PROGRAM C25_MC2AxisDriversCtrl
VAR
	fbMC2AxisCtrl		:  FB_MC2_AX5000AxisCtrl;

	stAxisConfig		: ST_AXIS_Config;	(*Has to be defined in Machine Config structure to retain data*)

	bStationHomed		: BOOL;
	bSeqHomingRequest	: BOOL;
	bSeqInProgress		: BOOL;

(*dummy sturcture to be replaced by global MC struct once implemnted*)
{library private}
	nAxis00TorqueLimitation								: UINT	:=	32767;
	nAxis00ActualTorque								 : INT;
	refAxis00											: AXIS_REF;
END_VAR

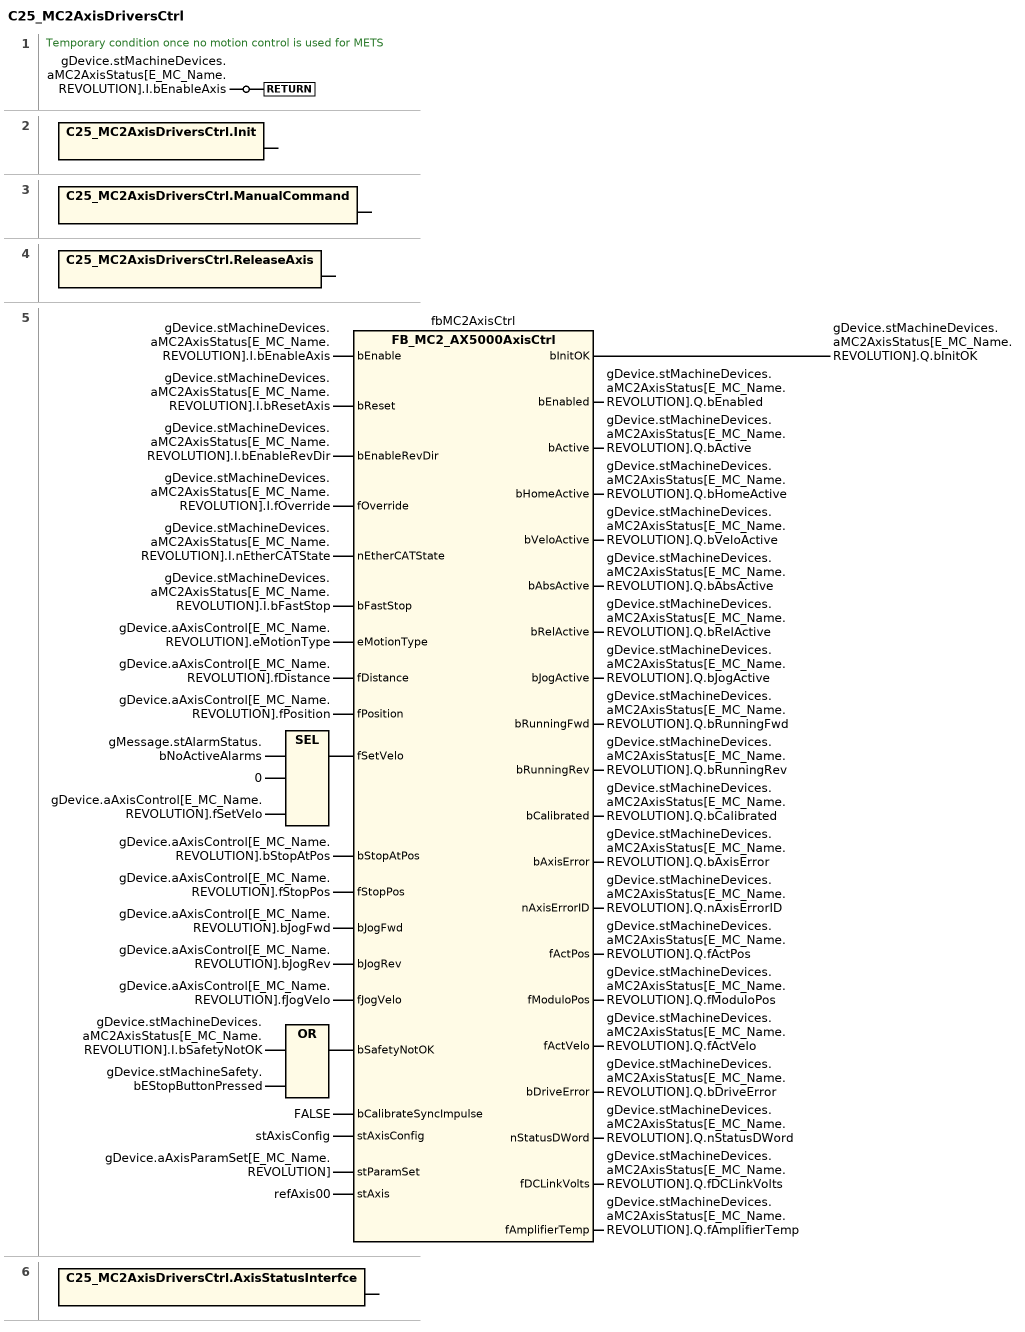
// NETWORK 1
// Temporary condition once no motion control is used for METS
IF NOT gDevice.stMachineDevices.aMC2AxisStatus[E_MC_Name.REVOLUTION].I.bEnableAxis THEN RETURN; END_IF

// NETWORK 2
C25_MC2AxisDriversCtrl.Init();

// NETWORK 3
C25_MC2AxisDriversCtrl.ManualCommand();

// NETWORK 4
C25_MC2AxisDriversCtrl.ReleaseAxis();

// NETWORK 5
fbMC2AxisCtrl(
    bEnable := gDevice.stMachineDevices.aMC2AxisStatus[E_MC_Name.REVOLUTION].I.bEnableAxis,
    bReset := gDevice.stMachineDevices.aMC2AxisStatus[E_MC_Name.REVOLUTION].I.bResetAxis,
    bEnableRevDir := gDevice.stMachineDevices.aMC2AxisStatus[E_MC_Name.REVOLUTION].I.bEnableRevDir,
    fOverride := gDevice.stMachineDevices.aMC2AxisStatus[E_MC_Name.REVOLUTION].I.fOverride,
    nEtherCATState := gDevice.stMachineDevices.aMC2AxisStatus[E_MC_Name.REVOLUTION].I.nEtherCATState,
    bFastStop := gDevice.stMachineDevices.aMC2AxisStatus[E_MC_Name.REVOLUTION].I.bFastStop,
    eMotionType := gDevice.aAxisControl[E_MC_Name.REVOLUTION].eMotionType,
    fDistance := gDevice.aAxisControl[E_MC_Name.REVOLUTION].fDistance,
    fPosition := gDevice.aAxisControl[E_MC_Name.REVOLUTION].fPosition,
    fSetVelo := SEL(gMessage.stAlarmStatus.bNoActiveAlarms, 0, gDevice.aAxisControl[E_MC_Name.REVOLUTION].fSetVelo),
    bStopAtPos := gDevice.aAxisControl[E_MC_Name.REVOLUTION].bStopAtPos,
    fStopPos := gDevice.aAxisControl[E_MC_Name.REVOLUTION].fStopPos,
    bJogFwd := gDevice.aAxisControl[E_MC_Name.REVOLUTION].bJogFwd,
    bJogRev := gDevice.aAxisControl[E_MC_Name.REVOLUTION].bJogRev,
    fJogVelo := gDevice.aAxisControl[E_MC_Name.REVOLUTION].fJogVelo,
    bSafetyNotOK := gDevice.stMachineDevices.aMC2AxisStatus[E_MC_Name.REVOLUTION].I.bSafetyNotOK OR gDevice.stMachineSafety.bEStopButtonPressed,
    bCalibrateSyncImpulse := FALSE,
    stAxisConfig := stAxisConfig,
    stParamSet := gDevice.aAxisParamSet[E_MC_Name.REVOLUTION],
    stAxis := refAxis00,
    bEnabled => gDevice.stMachineDevices.aMC2AxisStatus[E_MC_Name.REVOLUTION].Q.bEnabled,
    bActive => gDevice.stMachineDevices.aMC2AxisStatus[E_MC_Name.REVOLUTION].Q.bActive,
    bHomeActive => gDevice.stMachineDevices.aMC2AxisStatus[E_MC_Name.REVOLUTION].Q.bHomeActive,
    bVeloActive => gDevice.stMachineDevices.aMC2AxisStatus[E_MC_Name.REVOLUTION].Q.bVeloActive,
    bAbsActive => gDevice.stMachineDevices.aMC2AxisStatus[E_MC_Name.REVOLUTION].Q.bAbsActive,
    bRelActive => gDevice.stMachineDevices.aMC2AxisStatus[E_MC_Name.REVOLUTION].Q.bRelActive,
    bJogActive => gDevice.stMachineDevices.aMC2AxisStatus[E_MC_Name.REVOLUTION].Q.bJogActive,
    bRunningFwd => gDevice.stMachineDevices.aMC2AxisStatus[E_MC_Name.REVOLUTION].Q.bRunningFwd,
    bRunningRev => gDevice.stMachineDevices.aMC2AxisStatus[E_MC_Name.REVOLUTION].Q.bRunningRev,
    bCalibrated => gDevice.stMachineDevices.aMC2AxisStatus[E_MC_Name.REVOLUTION].Q.bCalibrated,
    bAxisError => gDevice.stMachineDevices.aMC2AxisStatus[E_MC_Name.REVOLUTION].Q.bAxisError,
    nAxisErrorID => gDevice.stMachineDevices.aMC2AxisStatus[E_MC_Name.REVOLUTION].Q.nAxisErrorID,
    fActPos => gDevice.stMachineDevices.aMC2AxisStatus[E_MC_Name.REVOLUTION].Q.fActPos,
    fModuloPos => gDevice.stMachineDevices.aMC2AxisStatus[E_MC_Name.REVOLUTION].Q.fModuloPos,
    fActVelo => gDevice.stMachineDevices.aMC2AxisStatus[E_MC_Name.REVOLUTION].Q.fActVelo,
    bDriveError => gDevice.stMachineDevices.aMC2AxisStatus[E_MC_Name.REVOLUTION].Q.bDriveError,
    nStatusDWord => gDevice.stMachineDevices.aMC2AxisStatus[E_MC_Name.REVOLUTION].Q.nStatusDWord,
    fDCLinkVolts => gDevice.stMachineDevices.aMC2AxisStatus[E_MC_Name.REVOLUTION].Q.fDCLinkVolts,
    fAmplifierTemp => gDevice.stMachineDevices.aMC2AxisStatus[E_MC_Name.REVOLUTION].Q.fAmplifierTemp); // FB_MC2_AX5000AxisCtrl
gDevice.stMachineDevices.aMC2AxisStatus[E_MC_Name.REVOLUTION].Q.bInitOK := fbMC2AxisCtrl.bInitOK;

// NETWORK 6
C25_MC2AxisDriversCtrl.AxisStatusInterfce();

ACTION AxisStatusInterfce:
//{warning 'CONVERSION MESSAGE: This text contained unprintable characters, that have been deleted'.}
gHMI.aAxisStatusHMI[E_MC_Name.REVOLUTION].bInitOK:=gDevice.stMachineDevices.aMC2AxisStatus[E_MC_Name.REVOLUTION].Q.bInitOK;
gHMI.aAxisStatusHMI[E_MC_Name.REVOLUTION].bEnabled:= gDevice.stMachineDevices.aMC2AxisStatus[E_MC_Name.REVOLUTION].Q.bEnabled;
gHMI.aAxisStatusHMI[E_MC_Name.REVOLUTION].bHomeActive :=   gDevice.stMachineDevices.aMC2AxisStatus[E_MC_Name.REVOLUTION].Q.bHomeActive;
gHMI.aAxisStatusHMI[E_MC_Name.REVOLUTION].bVeloActive:=gDevice.stMachineDevices.aMC2AxisStatus[E_MC_Name.REVOLUTION].Q.bVeloActive;
gHMI.aAxisStatusHMI[E_MC_Name.REVOLUTION].bRelativeActive:= gDevice.stMachineDevices.aMC2AxisStatus[E_MC_Name.REVOLUTION].Q.bRelActive;
gHMI.aAxisStatusHMI[E_MC_Name.REVOLUTION].bAbsoluteActive:= gDevice.stMachineDevices.aMC2AxisStatus[E_MC_Name.REVOLUTION].Q.bAbsActive;
gHMI.aAxisStatusHMI[E_MC_Name.REVOLUTION].bJogActive:= gDevice.stMachineDevices.aMC2AxisStatus[E_MC_Name.REVOLUTION].Q.bJogActive;

gHMI.aAxisStatusHMI[E_MC_Name.REVOLUTION].eMotionState := refAxis00.Status.MotionState;

gHMI.aAxisStatusHMI[E_MC_Name.REVOLUTION].bOperational 	:=refAxis00.Status.Operational;
gHMI.aAxisStatusHMI[E_MC_Name.REVOLUTION].bHomed 	:=refAxis00.Status.Homed;
gHMI.aAxisStatusHMI[E_MC_Name.REVOLUTION].bHasJob	:=refAxis00.Status.HasJob;
gHMI.aAxisStatusHMI[E_MC_Name.REVOLUTION].bHomingBusy 	:=refAxis00.Status.HomingBusy;
gHMI.aAxisStatusHMI[E_MC_Name.REVOLUTION].bNotMoving 	:=refAxis00.Status.NotMoving;
gHMI.aAxisStatusHMI[E_MC_Name.REVOLUTION].bInTargetPosition 	:=refAxis00.Status.InTargetPosition;
gHMI.aAxisStatusHMI[E_MC_Name.REVOLUTION].bMovingPositiveDirection 	:=refAxis00.Status.PositiveDirection;
gHMI.aAxisStatusHMI[E_MC_Name.REVOLUTION].bMovingNegativeDirection	:=refAxis00.Status.NegativeDirection;
gHMI.aAxisStatusHMI[E_MC_Name.REVOLUTION].bInPositionRange 	:=refAxis00.Status.InPositionArea;
gHMI.aAxisStatusHMI[E_MC_Name.REVOLUTION].bError 	:=	refAxis00.Status.Error;
gHMI.aAxisStatusHMI[E_MC_Name.REVOLUTION].nErrorId 	:= refAxis00.Status.ErrorID;

gHMI.aAxisStatusHMI[E_MC_Name.REVOLUTION].fActualPosition :=refAxis00.NcToPlc.ModuloActPos;
gHMI.aAxisStatusHMI[E_MC_Name.REVOLUTION].fActualVelocity :=refAxis00.NcToPlc.ActVelo;
gHMI.aAxisStatusHMI[E_MC_Name.REVOLUTION].fSetpointPosition :=refAxis00.NcToPlc.ModuloSetPos;

(****************************************************************************************************************************************)
(****************************************************************************************************************************************)
(****************************************************************************************************************************************)
END_ACTION

ACTION Init:
gDevice.stMachineDevices.aMC2AxisStatus[E_MC_Name.REVOLUTION].I.bEnableRevDir 	:= TRUE;
gDevice.stMachineDevices.aMC2AxisStatus[E_MC_Name.REVOLUTION].I.fOverride	:= 100;
gDevice.stMachineDevices.aMC2AxisStatus[E_MC_Name.REVOLUTION].I.nEtherCATState	:= 8;

nAxis00TorqueLimitation := stAxisConfig.nTorqueLimitation;
END_ACTION

ACTION ManualCommand:
IF NOT gDevice.stMetsStatus.stMachineMode.bManual	THEN
	RETURN;
END_IF

gDevice.stMachineDevices.aMC2AxisStatus[E_MC_Name.REVOLUTION].I.bEnableAxis := gHMI.aAxisCtrlHMI[E_MC_Name.REVOLUTION].stReqEanble.bButtonState;
gDevice.stMachineDevices.aMC2AxisStatus[E_MC_Name.REVOLUTION].I.bResetAxis := gHMI.aAxisCtrlHMI[E_MC_Name.REVOLUTION].stReqReset.bButtonState;

IF NOT bSeqInProgress	THEN
	gDevice.aAxisControl[E_MC_Name.REVOLUTION].eMotionType := gHMI.aAxisCtrlHMI[E_MC_Name.REVOLUTION].eMotionType;

	gDevice.aAxisControl[E_MC_Name.REVOLUTION].bJogFwd := gHMI.aAxisCtrlHMI[E_MC_Name.REVOLUTION].stReqJogFwd.bButtonState;
	gDevice.aAxisControl[E_MC_Name.REVOLUTION].bJogRev := gHMI.aAxisCtrlHMI[E_MC_Name.REVOLUTION].stReqJogRev.bButtonState;
	gDevice.aAxisControl[E_MC_Name.REVOLUTION].fJogVelo	:= gHMI.aAxisCtrlHMI[E_MC_Name.REVOLUTION].fJogVelocity;

	gDevice.aAxisControl[E_MC_Name.REVOLUTION].fDistance := gHMI.aAxisCtrlHMI[E_MC_Name.REVOLUTION].fDistance;
	gDevice.aAxisControl[E_MC_Name.REVOLUTION].fPosition := gHMI.aAxisCtrlHMI[E_MC_Name.REVOLUTION].fPosition;
	gDevice.aAxisControl[E_MC_Name.REVOLUTION].fSetVelo := gHMI.aAxisCtrlHMI[E_MC_Name.REVOLUTION].fVelocity;

	gDevice.aAxisControl[E_MC_Name.REVOLUTION].bStopAtPos	 := gHMI.aAxisCtrlHMI[E_MC_Name.REVOLUTION].bStopAtPos;
	gDevice.aAxisControl[E_MC_Name.REVOLUTION].fStopPos	 := gHMI.aAxisCtrlHMI[E_MC_Name.REVOLUTION].fStopPos;

	IF gHMI.aAxisCtrlHMI[E_MC_Name.REVOLUTION].stReqPositioning.bButtonState THEN
	
		gDevice.aAxisControl[E_MC_Name.REVOLUTION].eMotionType 	:= E_AXIS_MotionType.MCHOME;
	END_IF
END_IF

IF bStationHomed	AND
	gDevice.stMachineDevices.aMC2AxisStatus[E_MC_Name.REVOLUTION].Q.bActive 	THEN

		bStationHomed				:=	FALSE;
		bSeqHomingRequest			:=	TRUE;
END_IF
END_ACTION

ACTION ReleaseAxis:
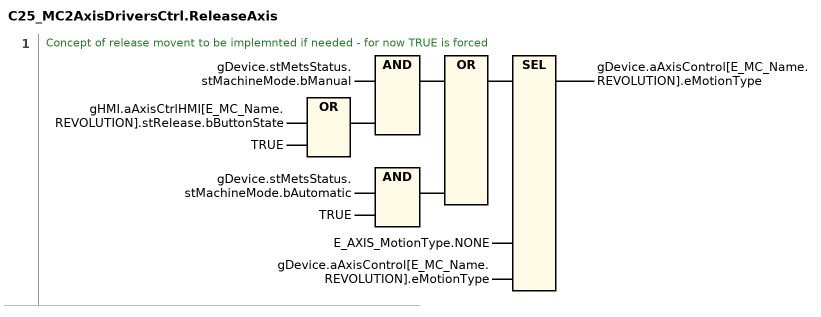
// NETWORK 1
// Concept of release movent to be implemnted if needed - for now TRUE is forced
gDevice.aAxisControl[E_MC_Name.REVOLUTION].eMotionType := SEL(gDevice.stMetsStatus.stMachineMode.bManual AND (gHMI.aAxisCtrlHMI[E_MC_Name.REVOLUTION].stRelease.bButtonState OR TRUE) OR gDevice.stMetsStatus.stMachineMode.bAutomatic AND TRUE, E_AXIS_MotionType.NONE, gDevice.aAxisControl[E_MC_Name.REVOLUTION].eMotionType);
END_ACTION

END_PROGRAM

(* stored: Version 1.1.0.1
   POU C25_MC2AxisDriversCtrl: Id {71d8f4d4-9a86-42cf-94d1-0baa13f4486b}, SpecialFunc None
   Action AxisStatusInterfce: Id {c9e7b0c1-cc69-438c-913f-de2e60ad22af}
   Action Init: Id {2a8388d1-baae-4e7f-b2d6-041023c6e58a}
   Action ManualCommand: Id {be234cb4-fb97-40b6-8a93-66ea8e64cec0}
   Action ReleaseAxis: Id {7db3d204-6f7f-4d60-87b8-0255b90e5d49} *)
